(* IEC 61131-3 sources: POMIRTS_lab3/AS/Library/IF361, 3 files *)

(* ---- IF361.typ ---- *)
(********************************************************************
 * COPYRIGHT (C) BERNECKER + RAINER, AUSTRIA, A-5142 EGGELSBERG
 ********************************************************************
 * Library: IF361
 * File: IF361.typ
 * Created: 11.11.2003
 ********************************************************************
 * Global data types of library IF361
 ********************************************************************)
TYPE
	if361_IfCfg : STRUCT
		idle	: UINT ;
		delime	: UINT ;
		delim	: ARRAY[0..1] OF USINT ;
		tx_cnt	: UINT ;
		rx_cnt	: UINT ;
		tx_len	: UINT ;
		rx_len	: UINT ;
		argc	: UINT ;
		argv	: UDINT ;
	END_STRUCT;
	if361_Iop : STRUCT
		io_type	: USINT ;
		master_no	: USINT ;
		slave_no	: USINT ;
		module_adr	: USINT ;
		intern_off	: USINT ;
		mode	: USINT ;
		datalen	: USINT ;
		reserve	: USINT ;
		data_adr	: UDINT ;
	END_STRUCT;
	if361_l2dp : STRUCT
		baudrate	: UINT ;
		station	: USINT ;
		freeze	: USINT ;
		sync	: USINT ;
		glob_cont	: USINT ;
		data_exchg	: USINT ;
	END_STRUCT;
END_TYPE

(* ---- IF361.fun ---- *)
(********************************************************************
 * COPYRIGHT (C) BERNECKER + RAINER, AUSTRIA, A-5142 EGGELSBERG
 ********************************************************************
 * Library: IF361
 * File: IF361.fun
 * Created: 11.11.2003
 ********************************************************************
 * Functions and function blocks of library IF361
 ********************************************************************)
FUNCTION_BLOCK IF361_frm_rdwr
	VAR_INPUT
		pSend	:UDINT;
		sendlng	:USINT;
		cmd	:USINT;
		ident	:UDINT;
		pRec	:UDINT;
	END_VAR
	VAR_OUTPUT
		rec_lng	:USINT;
		status	:UINT;
	END_VAR
	VAR
		statusro	:UINT;
		retry	:USINT;
		WR_buflng	:UINT;
		WR_buffer	:UDINT;
		frm_step	:USINT;
		bufferdat	:REFERENCE TO USINT;
		zzFRM_gbuf00000	:FRM_gbuf;
		zzFRM_write00001	:FRM_write;
		zzFRM_robuf00002	:FRM_robuf;
		zzFRM_read00003	:FRM_read;
		zzFRM_rbuf00004	:FRM_rbuf;
	END_VAR
END_FUNCTION_BLOCK
FUNCTION_BLOCK IF361
	VAR_INPUT
		enable	:BOOL;
		device	:UDINT;
		L2DPpara	:REFERENCE TO if361_l2dp;
		outbuf	:UDINT;
		outlen	:UDINT;
		inbuf	:UDINT;
		inlen	:UDINT;
		outcopy	:REFERENCE TO BOOL;
		incopy	:REFERENCE TO BOOL;
	END_VAR
	VAR_OUTPUT
		status	:UINT;
	END_VAR
	VAR
		bufcleared	:BOOL;
		chg_statio	:BOOL;
		station	:USINT;
		leave_loop	:BOOL;
		userstatus	:USINT;
		exit	:BOOL;
		frmoffset	:USINT;
		leave_send	:BOOL;
		blockoffse	:USINT;
		newblock	:BOOL;
		offset	:USINT;
		to_sendlng	:USINT;
		output	:USINT;
		input	:USINT;
		i_len	:USINT;
		o_len	:USINT;
		reclen	:USINT;
		rec	:USINT;
		frm	:IF361_frm_rdwr;
		send	:USINT;
		sendlng	:USINT;
		cmd	:USINT;
		buffsize	:UINT;
		diag_data_	:USINT;
		param_data	:USINT;
		CFG_dataLen	:USINT;
		wait_loop	:USINT;
		valuewr	:UINT;
		ident	:UDINT;
		baudrate	:UDINT;
		ifcfg	:if361_IfCfg;
		valuerd	:UINT;
		ioident	:UDINT;
		src	:USINT;
		Kennung	:UINT;
		iop	:if361_Iop;
		baudfrm	:UINT;
		baud	:UINT;
		slot	:USINT;
		SubSlot	:USINT;
		interface	:USINT;
		Slot	:USINT;
		length	:UINT;
		i	:USINT;
		exchange	:BOOL;
		chg_buffer	:BOOL;
		u_step	:USINT;
		outLEN	:USINT;
		inLEN	:USINT;
		allocated	:UDINT;
		cmp_buf	:UDINT;
		L2DPstep	:USINT;
		SYS_initcn	:UDINT;
		initcnt	:UDINT;
		devicestr	:REFERENCE TO USINT;
		tosend	:REFERENCE TO USINT;
		oldsend	:REFERENCE TO USINT;
		zzIO_mphydef00000	:IO_mphydef;
		zzIO_data00001	:IO_data;
		zzIO_mphydef00002	:IO_mphydef;
		zzIO_data00003	:IO_data;
		zzIO_mphydef00004	:IO_mphydef;
		zzIO_data00005	:IO_data;
		zzFRM_xopen00006	:FRM_xopen;
		zzIO_mphydef00007	:IO_mphydef;
		zzIO_data00008	:IO_data;
		zzIO_mphydef00009	:IO_mphydef;
		avtident	:UDINT;
		null_after_dl	:BOOL;
		avt_status	:UINT;
		avtinfo	:UDINT;
		avtname	:USINT;
		zzFRM_xopen00000	:FRM_xopen;
		zzIO_mphydef00001	:IO_mphydef;
		zzIO_data00002	:IO_data;
		zzIO_mphydef00003	:IO_mphydef;
		zzIO_data00004	:IO_data;
		zzIO_mphydef00005	:IO_mphydef;
		zzIO_data00006	:IO_data;
		zzFRM_xopen00007	:FRM_xopen;
		zzIO_mphydef00008	:IO_mphydef;
		zzIO_data00009	:IO_data;
		zzIO_mphydef00010	:IO_mphydef;
		hochlauf_flag	:BOOL;
	END_VAR
END_FUNCTION_BLOCK

(* ---- IF361.var ---- *)
(********************************************************************
 * COPYRIGHT (C) BERNECKER + RAINER, AUSTRIA, A-5142 EGGELSBERG
 ********************************************************************
 * Library: IF361
 * File: IF361.var
 * Created: 11.11.2003
 ********************************************************************
 * Constants of library IF361
 ********************************************************************)
VAR CONSTANT
	ERR_IF361_RESTART_AT_BAUDCHANGE	: UINT	:= 12070;
	ERR_IF361_RDWR_NO_FRAMESTART	: UINT	:= 12055;
	ERR_IF361_WAIT_FOR_DATAMODE	: UINT	:= 12079;
	ERR_IF361_OTHER_MASTER_CFG	: UINT	:= 12072;
	ERR_IF361_COMMAND_INVALID	: UINT	:= 12080;
	ERR_IF361_RDWR_WRONG_PTR	: UINT	:= 12051;
	ERR_IF361_RDWR_NO_ANSWER	: UINT	:= 12056;
	ERR_IF361_PARAM_CONFLICT	: UINT	:= 12073;
	ERR_IF361_FRAME_TOO_LONG	: UINT	:= 12050;
	ERR_IF361_SLAVE_OFFLINE	: UINT	:= 12076;
	ERR_IF361_PARAM_INVALID	: UINT	:= 12081;
	ERR_IF361_DEVICE_STRING	: UINT	:= 12058;
	ERR_IF361_ANSWER_LENGTH	: UINT	:= 12071;
	ERR_IF361_SPC3LESS_MEM	: UINT	:= 12082;
	ERR_IF361_SPC3DOUT_LEN	: UINT	:= 12085;
	ERR_IF361_SPC3DIAG_LEN	: UINT	:= 12086;
	ERR_IF361_SETTING_BAUD	: UINT	:= 12057;
	ERR_IF361_RDWR_NO_DATA	: UINT	:= 12054;
	ERR_IF361_L2DPPARA_PTR	: UINT	:= 12066;
	ERR_IF361_SPC3SYS_INI	: UINT	:= 12092;
	ERR_IF361_SPC3PRM_LEN	: UINT	:= 12087;
	ERR_IF361_SPC3INV_LEN	: UINT	:= 12090;
	ERR_IF361_SPC3INV_CHK	: UINT	:= 12091;
	ERR_IF361_SPC3DIN_LEN	: UINT	:= 12084;
	ERR_IF361_SPC3CFG_LEN	: UINT	:= 12088;
	ERR_IF361_INV_WRAPCNT	: UINT	:= 12093;
	ERR_IF361_INV_BYTECNT	: UINT	:= 12094;
	ERR_IF361_WRONG_BAUD	: UINT	:= 12067;
	ERR_IF361_SPC3INVADR	: UINT	:= 12097;
	ERR_IF361_SPC3BLKPRG	: UINT	:= 12096;
	ERR_IF361_SPC3BLKDEL	: UINT	:= 12095;
	ERR_IF361_OUTBUF_PTR	: UINT	:= 12059;
	ERR_IF361_SUBSLOTNR	: UINT	:= 12064;
	ERR_IF361_STATIONNR	: UINT	:= 12078;
	ERR_IF361_INTERFACE	: UINT	:= 12063;
	ERR_IF361_INBUF_PTR	: UINT	:= 12060;
	ERR_IF361_WATCHDOG	: UINT	:= 12077;
	ERR_IF361_SPC3NOFF	: UINT	:= 12083;
	ERR_IF361_NO_IF361	: UINT	:= 12068;
	ERR_IF361_INOUTLEN	: UINT	:= 12069;
	ERR_IF361_SLOTNR	: UINT	:= 12065;
	ERR_IF361_OUTLEN	: UINT	:= 12061;
	ERR_IF361_INLEN	: UINT	:= 12062;
END_VAR
